Omron CX-Programmer project NewProject (CX-Programmer 9.51)

# PLC My_first_project: CP1L L
; This is my first LD project

## Global symbols (name address type ; comment)
0.00 BOOL  ; Input
100.00 BOOL  ; output

## Program NewProgram1 (cyclic task 0)
Local symbols
btn_1 0.00 BOOL  ; Comment
btn_2 0.01 BOOL  ; Comment
btn_3 0.02 BOOL  ; Comment

### Section Section1

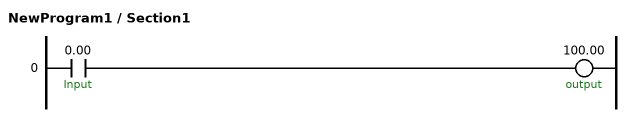
; rung 0
LD 0.00  ; Input
OUT 100.00  ; output

### Section END
; rung 0
END(001)